// Setup Arm Base Controller, Hold at Current Posture
FUNCTION_BLOCK FB_SetupArmCtrlBase IMPLEMENTS I_SetupArmCtrl
VAR_INPUT
END_VAR
VAR_OUTPUT
END_VAR
VAR
	// flag if the controller has finished all its jobs
	m_isFinished:BOOL:=FALSE;
	
	// controller execute time period
	m_timePeriod :LREAL:=0;
	
	// arm control data
	m_cmdJntPos : VEC5d;
	m_cmdJntVel : VEC5d;
	m_cmdJntAcc : VEC5d;
	m_cmdJntTrq : VEC5d;
	m_jntOPMode : Vec5i;
	m_jntEnableFlag :Vec5i;
END_VAR

// override this function in each exact controller
METHOD PROTECTED calcCmdJntPos : BOOL
VAR_IN_OUT CONSTANT
	i_setupArm	:FB_SetupArm;
END_VAR
END_METHOD

// override this function in each exact controller
METHOD PROTECTED calcCmdJntTrq : BOOL
VAR_IN_OUT CONSTANT
	i_setupArm	:FB_SetupArm;
END_VAR
// set joint torque to zero in default
m_cmdJntTrq := g_zeroVec5d;
END_METHOD

// override this function in each exact controller
// NOTICE: set joint control mode here, and do some initialization if needed
METHOD PUBLIC init : BOOL
VAR_IN_OUT CONSTANT
	i_setupArm	:FB_SetupArm;
END_VAR
VAR_IN_OUT 
	r_setupArmCtrlCmd :ST_SetupArmCtrlCmds;
END_VAR
m_timePeriod:=0;
m_jntEnableFlag :=g_zeroVec5i;// setup arm joint is off by default
m_jntOPMode:=g_setupAllPosMode;
m_cmdJntPos:=i_setupArm.curJntPos;
m_cmdJntVel:=g_zeroVec5d;
m_cmdJntAcc:=g_zeroVec5d;
m_cmdJntTrq:=g_zeroVec5d;

// update commands to arm
r_setupArmCtrlCmd.m_jntEnableFlag :=m_jntEnableFlag;
r_setupArmCtrlCmd.m_cmdJntPos:=m_cmdJntPos;
r_setupArmCtrlCmd.m_cmdJntVel:=m_cmdJntVel;
r_setupArmCtrlCmd.m_cmdJntAcc:=m_cmdJntAcc;
r_setupArmCtrlCmd.m_cmdJntTrq:=m_cmdJntTrq;
r_setupArmCtrlCmd.m_jntOPMode:=m_jntOPMode;
END_METHOD

PROPERTY isFinished : BOOL
GET
isFinished:=m_isFinished;
END_GET
END_PROPERTY

{warning '添加方法实现'}
METHOD reset : BOOL
m_isFinished:=FALSE;
m_timePeriod:=0;
END_METHOD

{warning '添加方法实现'}
METHOD run : BOOL
VAR_IN_OUT CONSTANT
	i_setupArm	:FB_SetupArm;
END_VAR
VAR_IN_OUT 
	r_setupArmCtrlCmd :ST_SetupArmCtrlCmds;
END_VAR

VAR
	i:INT;
END_VAR
IF m_isFinished THEN
	RETURN;
END_IF

// check if arm enabled
IF FALSE = i_setupArm.isEnabled(m_jntEnableFlag) THEN
//	RETURN;
END_IF

// calculate command joint position--Motion control
calcCmdJntPos(i_setupArm);

// calculate command joint torque -- Force control
calcCmdJntTrq(i_setupArm);

// update commands to arm
r_setupArmCtrlCmd.m_jntEnableFlag :=m_jntEnableFlag;
r_setupArmCtrlCmd.m_cmdJntPos:=m_cmdJntPos;
r_setupArmCtrlCmd.m_cmdJntVel:=m_cmdJntVel;
r_setupArmCtrlCmd.m_cmdJntAcc:=m_cmdJntAcc;
r_setupArmCtrlCmd.m_cmdJntTrq:=m_cmdJntTrq;
r_setupArmCtrlCmd.m_jntOPMode:=m_jntOPMode;

// update time period
m_timePeriod := m_timePeriod+g_slaveArmCtrlCycleTime;
END_METHOD

END_FUNCTION_BLOCK

(* stored: Version 1.1.0.1, ProductVersion 3.1.4024.12
   POU FB_SetupArmCtrlBase: Id {0b31894e-90eb-4625-a1b2-b64eb3714a74}, SpecialFunc None
   Method calcCmdJntPos: Id {93f4b4dc-c2f7-491d-8c73-da994ea2dbef}
   Method calcCmdJntTrq: Id {6ae77395-a816-419a-a1f1-e8f5e88f907c}
   Method init: Id {39abdba7-12c4-423b-9680-dbfc1169a913}
   Property isFinished: Id {1ba11897-c13c-426e-b2eb-85c7dda0df9b}
   Get Get: Id {90cfe719-a7f9-4e4f-9a72-5775b0006367}
   Method reset: Id {90707f36-a1c9-4b9c-b59d-3c71748b414a}
   Method run: Id {08326719-dfd7-43d5-bd4f-6865187be57d} *)
